// TwinCAT 3 PLC project PLC_Ladder_Hardware_Integration
// ProgramVersion: 3.1.4024.0
// CompilerDefines: VISU_USEWSTRING
// libraries:
//   Tc2_Math, * (Beckhoff Automation GmbH)
//   Tc2_MC2, * (Beckhoff Automation GmbH)
//   Tc2_NC, * (Beckhoff Automation GmbH)
//   Tc2_Standard, * (Beckhoff Automation GmbH)
//   Tc2_System, * (Beckhoff Automation GmbH)
//   Tc2_Utilities, * (Beckhoff Automation GmbH)
//   Tc3_Module, * (Beckhoff Automation GmbH)
// project tree:
//   / GlobalTextList.TcGTLO (not stored), PlcTask.TcTTO, Visualization Manager.TcVMO (not stored)
//   GVLs/ GVL.TcGVL (not stored), GVLLD.TcGVL
//   POUs/ MAIN.TcPOU (not stored), ladder_logic_diagram.TcPOU, Meters_Travelled.TcPOU (not stored), SYSTEM.TcPOU (not stored), Safety_Zones.TcDUT (not stored)
//   VISUs/ Charge_Velocity_Distance.TcVIS (not stored), Header.TcVIS (not stored), ImagePool.TcIPO (not stored), log_file.TcVIS, MainScreen.TcVIS (not stored), Nav.TcVIS, Nav_1.TcVIS, Safty_Zones_and_Modes.TcVIS (not stored)
// real-time tasks:
//   TASK PlcTask: cycle T#10ms, priority 20, ADS port 350
//   TASK VISU_TASK: cycle T#200000us, priority 30, ADS port 351
// motion (NC):
//   TASK NC-Task 1 SAF: cycle T#2ms, priority 4, ADS port 501
//   TASK NC-Task 1 SVB: cycle T#10ms, priority 8, ADS port 511
//   AXIS Axis 1 (id 1)
//     Dynamic: Acceleration=5067.48, Deceleration=5067.48, Jerk=23830.8
//     Velo: RefSearch=14.56175, RefSync=14.56175, SlowManual=72.80875, FastManual=436.8525, Fast=1456.175, Maximum=1456.17
//     TargetPosControl: Range=20
//     OtherSettings: AllowMotionCmdToSlave=true, PulseDistancePos=20, PulseDistanceNeg=20
//     encoder EncType=19
//       EncPara: ScaleFactorNumerator=15.7, ScaleFactorDenominator=1048576, Inverse=true, MaxCount=#xffffffff
//     drive DrvType=16
//       DrvPara: Inverse=true, MaxCount=#xffffffff
//         Analog: VeloReferenz=1601.7925, VeloScale=32, TorqueSetpointScale=10, ScaleFactorActTorque=0.1
//         TimeComp: TaskDelayCycles=1
//     controller CtrType=1
//       CtrPara: PriorControlFactor=1
//         PosDiffControl: Range=40000
//         Observer: BandWidth=20
//   AXIS Axis 2 (id 2)
//     Dynamic: Acceleration=5067.48, Deceleration=5067.48, Jerk=23830.8
//     Velo: RefSearch=14.56175, RefSync=14.56175, SlowManual=72.80875, FastManual=436.8525, Fast=1456.175, Maximum=1456.17
//     TargetPosControl: Range=20
//     OtherSettings: AllowMotionCmdToSlave=true, PulseDistancePos=20, PulseDistanceNeg=20
//     encoder EncType=19
//       EncPara: ScaleFactorNumerator=15.7, ScaleFactorDenominator=1048576, MaxCount=#xffffffff
//     drive DrvType=16
//       DrvPara: MaxCount=#xffffffff
//         Analog: VeloReferenz=1601.7925, VeloScale=32, TorqueSetpointScale=10, ScaleFactorActTorque=0.1
//         TimeComp: TaskDelayCycles=1
//     controller CtrType=1
//       CtrPara: PriorControlFactor=1
//         PosDiffControl: Range=40000
//         Observer: BandWidth=20
//   AXIS Axis 3 (id 3)
//     Dynamic: Acceleration=14588.3136, Deceleration=14588.3136, Jerk=43764.9408
//     Velo: RefSearch=97.255424, RefSync=97.255424, SlowManual=486.27712, FastManual=2917.66272, Fast=9725.5424, Maximum=9725.5424
//     OtherSettings: AllowMotionCmdToSlave=true
//     encoder EncType=19
//       EncPara: ScaleFactorNumerator=104.8576, ScaleFactorDenominator=1048576, MaxCount=#xffffffff
//     drive DrvType=16
//       DrvPara: MaxCount=#xffffffff
//         Analog: VeloReferenz=10698.09664, VeloScale=32, TorqueSetpointScale=10, ScaleFactorActTorque=0.1
//         TimeComp: TaskDelayCycles=1
//     controller CtrType=1
//       CtrPara: PriorControlFactor=1
//         PosDiffControl: Range=10
//         Observer: BandWidth=20
// variable links:
//   PLC_Ladder_Hardware_Integration/PLC_Ladder_Hardware_Integration Instance <-> NC-Task 1 SAF/Axes/Axis 1
//     PlcTask Inputs/MAIN.AxisB.NcToPlc <-> Outputs/ToPlc
//     PlcTask Outputs/MAIN.AxisB.PlcToNc <-> Inputs/FromPlc
//   PLC_Ladder_Hardware_Integration/PLC_Ladder_Hardware_Integration Instance <-> NC-Task 1 SAF/Axes/Axis 2
//     PlcTask Inputs/MAIN.AxisA.NcToPlc <-> Outputs/ToPlc
//     PlcTask Outputs/MAIN.AxisA.PlcToNc <-> Inputs/FromPlc

CONFIGURATION PLC_Ladder_Hardware_Integration
    RESOURCE PLC ON TwinCAT3
        TASK PlcTask(INTERVAL := T#10ms, PRIORITY := 20);
        PROGRAM ladder_logic_diagram WITH PlcTask : ladder_logic_diagram;
        PROGRAM MAIN WITH PlcTask : MAIN;
    END_RESOURCE
END_CONFIGURATION

// ---- GVLs/GVLLD.TcGVL
{attribute 'qualified_only'}
VAR_GLOBAL
	
//Input Variables 
ONOFF_Buton               AT %I* : BOOL;
Manual_Stop_Buton         AT %I* : BOOL;
Manual_Mode_Buton         AT %I* : BOOL;
Autonomous_Mode_Buton     AT %I* : BOOL;
Lock_Mode_Buton           AT %I* : BOOL;
Clear_Reset_Buton         AT %I* : BOOL;
Resume_Buton              AT %I* : BOOL;
view_safety               AT %I* : BOOL;


//Output Variables 
Brake                     AT %Q* : BOOL;  
Kontak                    AT %Q* : BOOL;
Front_White_Zone          AT %Q* : BOOL;
Front_Red_Zone            AT %Q* : BOOL;
Front_Purple_Zone         AT %Q* : BOOL;
Front_Grey_Pink_Zone      AT %Q* : BOOL;
Robot_Clear_Lidar         AT %Q* : BOOL;
Robot_Manual_Mode         AT %Q* : BOOL;
Robot_Autonomous_Mode     AT %Q* : BOOL;
Robot_Lock_Mode           AT %Q* : BOOL;
Robot_Mode_Run            AT %Q* : BOOL;
lift_up_Q                 AT %Q* : BOOL;
lift_down_Q            	  AT %Q* : BOOL;
zone_1                    AT %Q* : BOOL;
zone_2                    AT %Q* : BOOL;
zone_3                    AT %Q* : BOOL;
zone_4                    AT %Q* : BOOL;
zone_5                    AT %Q* : BOOL;
zone_6                    AT %Q* : BOOL;
auto_charge_signal        AT %Q* : BOOL;

//Memery Variables 

System_Trig               AT %M* : BOOL;
System_Set                AT %M* : BOOL;
Memory_Set		          AT %M* : BOOL;
White                     AT %M* : BOOL;
Red                       AT %M* : BOOL;
Purple                    AT %M* : BOOL;
Grey_Pink                 AT %M* : BOOL;
Lock_Mode_Reset           AT %M* : BOOL;
lift_up           		  AT %M* : BOOL;
lift_down				  AT %M* : BOOL;
lift_stop				  AT %M* : BOOL;
elavator_up				  AT %M* : BOOL;
elavator_down			  AT %M* : BOOL;
auto_charge_on            AT %M* : BOOL;
auto_charge_off           AT %M* : BOOL;
view_safety_state         AT %M* : BOOL;

first_time_read           AT %M* : BOOL;
second_time_read          AT %M* : BOOL;
END_VAR

// ---- POUs/ladder_logic_diagram.TcPOU
PROGRAM ladder_logic_diagram 
VAR
	t2s: TIME := TIME#3S;
	t0s: TIME := TIME#0S;
	Timer: TON;
	input : BOOL;
	output : BOOL; 
	TON_Reset: TON;
	TON_set: TON;
	TON_0: TON;
	TON_Trig: TON;
	TON_Autonomous: TON;
	TON_Manual: TON;
	TON_Lock: TON;
	Robot_Mode_Timer: TON;
	liftUP: TON;
	liftDOWN: TON;
	load_button  AT %I* : BOOL ;
	load_active AT %Q*: BOOL;
	trigger AT %M* : BOOL ;
	T: TIME;
	TON_1: TON;
	TON2: TON;
	TON_3: TON;
	activate_time_read: BOOL;
	TON_4: TON;
	second_read_triggered: BOOL;
	first_read_triggered: BOOL;
	TON_5: TON;
	TON_6: TON;
	TON_7: TON;
END_VAR
VAR // added by the converter: edge detectors and wires of the graphical bodies
    _rt1 : R_TRIG;
    _w1 : BOOL;
END_VAR

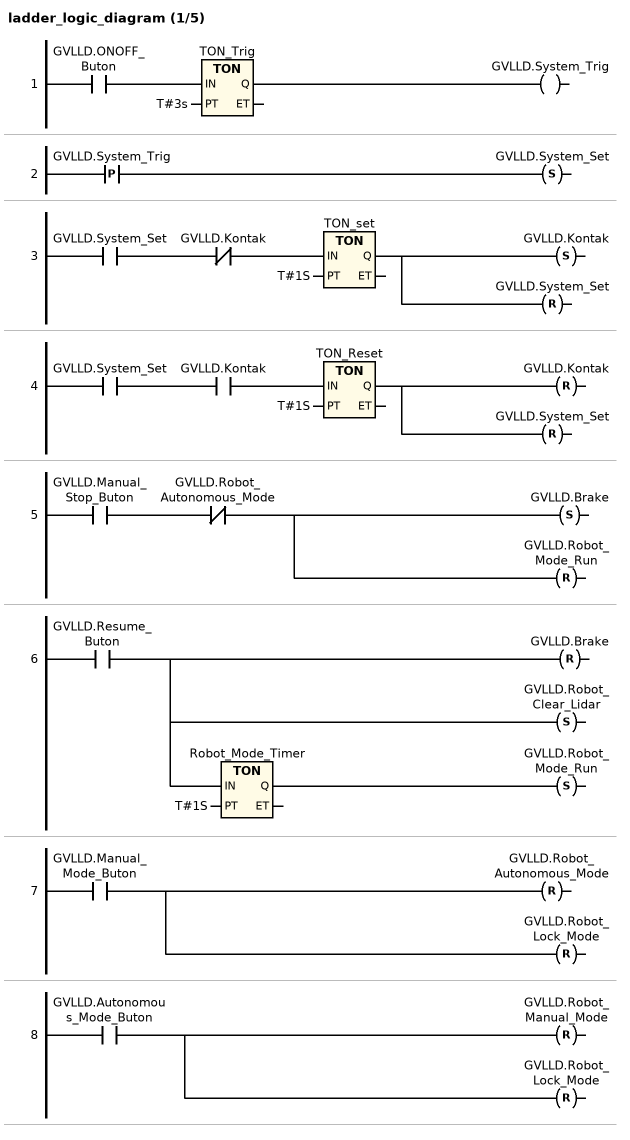
// NETWORK 1
TON_Trig(IN := GVLLD.ONOFF_Buton, PT := T#3s); // TON
GVLLD.System_Trig := TON_Trig.Q;

// NETWORK 2
_rt1(CLK := GVLLD.System_Trig);
GVLLD.System_Set S= _rt1.Q;

// NETWORK 3
TON_set(IN := GVLLD.System_Set AND NOT GVLLD.Kontak, PT := T#1S); // TON
GVLLD.Kontak S= TON_set.Q;
GVLLD.System_Set R= TON_set.Q;

// NETWORK 4
TON_Reset(IN := GVLLD.System_Set AND GVLLD.Kontak, PT := T#1S); // TON
GVLLD.Kontak R= TON_Reset.Q;
GVLLD.System_Set R= TON_Reset.Q;

// NETWORK 5
_w1 := GVLLD.Manual_Stop_Buton AND NOT GVLLD.Robot_Autonomous_Mode;
GVLLD.Brake S= _w1;
GVLLD.Robot_Mode_Run R= _w1;

// NETWORK 6
GVLLD.Brake R= GVLLD.Resume_Buton;
GVLLD.Robot_Clear_Lidar S= GVLLD.Resume_Buton;
Robot_Mode_Timer(IN := GVLLD.Resume_Buton, PT := T#1S); // TON
GVLLD.Robot_Mode_Run S= Robot_Mode_Timer.Q;

// NETWORK 7
GVLLD.Robot_Autonomous_Mode R= GVLLD.Manual_Mode_Buton;
GVLLD.Robot_Lock_Mode R= GVLLD.Manual_Mode_Buton;

// NETWORK 8
GVLLD.Robot_Manual_Mode R= GVLLD.Autonomous_Mode_Buton;
GVLLD.Robot_Lock_Mode R= GVLLD.Autonomous_Mode_Buton;

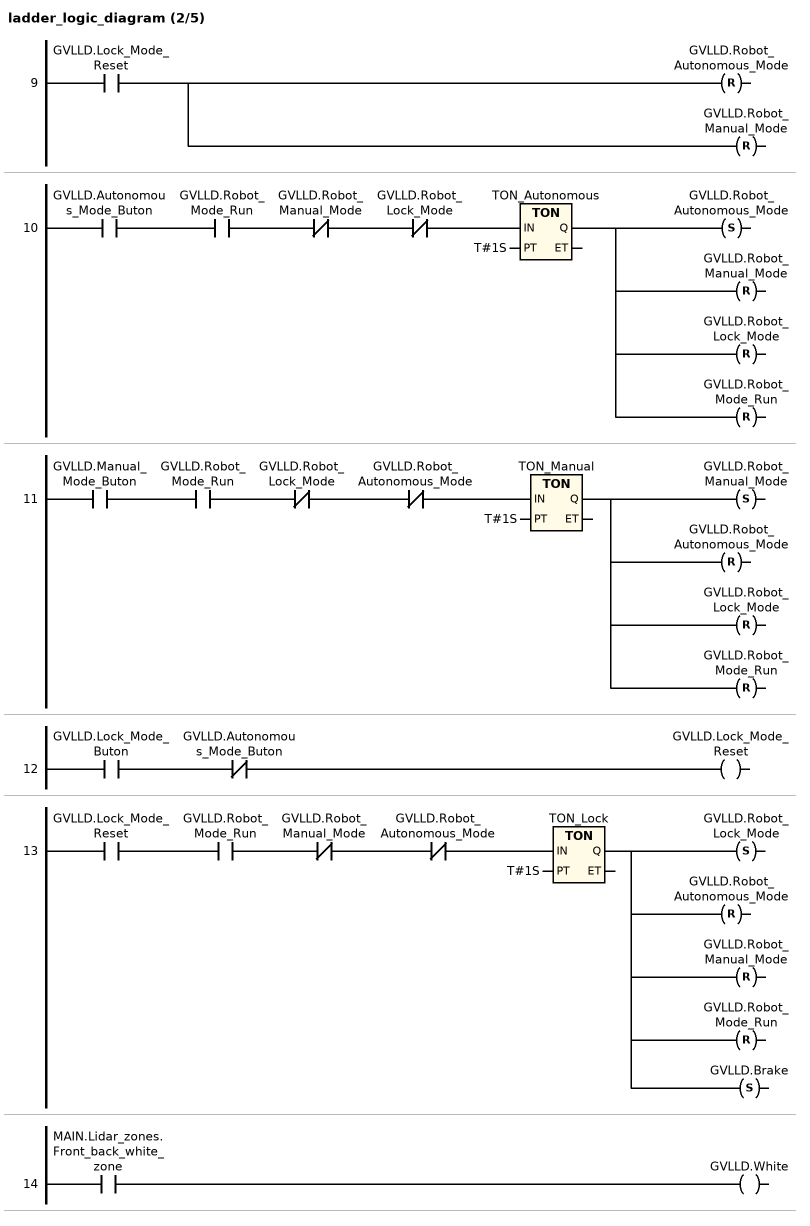
// NETWORK 9
GVLLD.Robot_Autonomous_Mode R= GVLLD.Lock_Mode_Reset;
GVLLD.Robot_Manual_Mode R= GVLLD.Lock_Mode_Reset;

// NETWORK 10
TON_Autonomous(IN := GVLLD.Autonomous_Mode_Buton AND GVLLD.Robot_Mode_Run AND NOT GVLLD.Robot_Manual_Mode AND NOT GVLLD.Robot_Lock_Mode, PT := T#1S); // TON
GVLLD.Robot_Autonomous_Mode S= TON_Autonomous.Q;
GVLLD.Robot_Manual_Mode R= TON_Autonomous.Q;
GVLLD.Robot_Lock_Mode R= TON_Autonomous.Q;
GVLLD.Robot_Mode_Run R= TON_Autonomous.Q;

// NETWORK 11
TON_Manual(IN := GVLLD.Manual_Mode_Buton AND GVLLD.Robot_Mode_Run AND NOT GVLLD.Robot_Lock_Mode AND NOT GVLLD.Robot_Autonomous_Mode, PT := T#1S); // TON
GVLLD.Robot_Manual_Mode S= TON_Manual.Q;
GVLLD.Robot_Autonomous_Mode R= TON_Manual.Q;
GVLLD.Robot_Lock_Mode R= TON_Manual.Q;
GVLLD.Robot_Mode_Run R= TON_Manual.Q;

// NETWORK 12
GVLLD.Lock_Mode_Reset := GVLLD.Lock_Mode_Buton AND NOT GVLLD.Autonomous_Mode_Buton;

// NETWORK 13
TON_Lock(IN := GVLLD.Lock_Mode_Reset AND GVLLD.Robot_Mode_Run AND NOT GVLLD.Robot_Manual_Mode AND NOT GVLLD.Robot_Autonomous_Mode, PT := T#1S); // TON
GVLLD.Robot_Lock_Mode S= TON_Lock.Q;
GVLLD.Robot_Autonomous_Mode R= TON_Lock.Q;
GVLLD.Robot_Manual_Mode R= TON_Lock.Q;
GVLLD.Robot_Mode_Run R= TON_Lock.Q;
GVLLD.Brake S= TON_Lock.Q;

// NETWORK 14
GVLLD.White := MAIN.Lidar_zones.Front_back_white_zone;

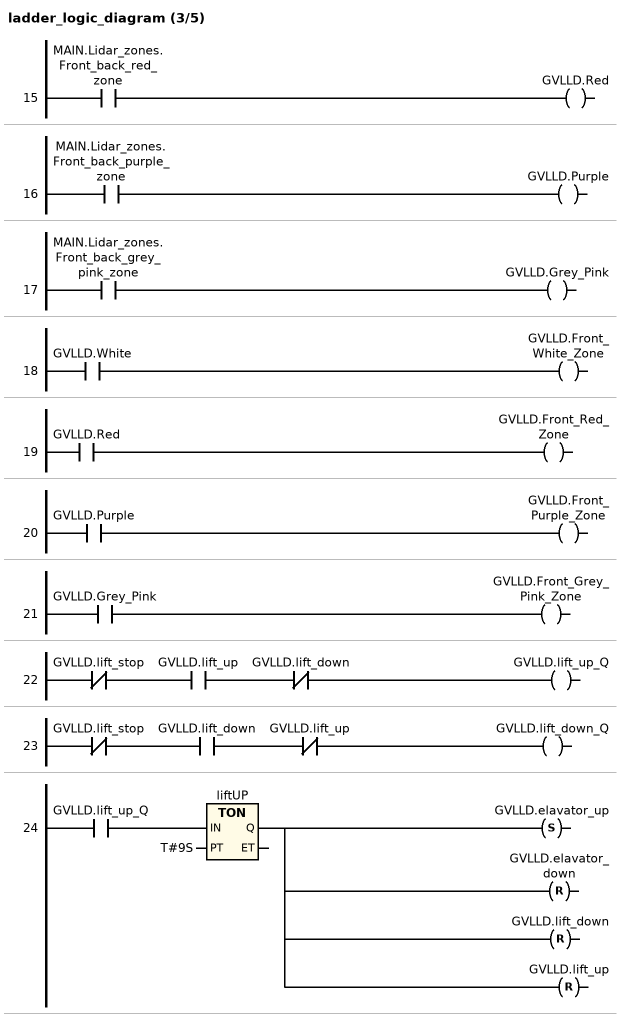
// NETWORK 15
GVLLD.Red := MAIN.Lidar_zones.Front_back_red_zone;

// NETWORK 16
GVLLD.Purple := MAIN.Lidar_zones.Front_back_purple_zone;

// NETWORK 17
GVLLD.Grey_Pink := MAIN.Lidar_zones.Front_back_grey_pink_zone;

// NETWORK 18
GVLLD.Front_White_Zone := GVLLD.White;

// NETWORK 19
GVLLD.Front_Red_Zone := GVLLD.Red;

// NETWORK 20
GVLLD.Front_Purple_Zone := GVLLD.Purple;

// NETWORK 21
GVLLD.Front_Grey_Pink_Zone := GVLLD.Grey_Pink;

// NETWORK 22
GVLLD.lift_up_Q := NOT GVLLD.lift_stop AND GVLLD.lift_up AND NOT GVLLD.lift_down;

// NETWORK 23
GVLLD.lift_down_Q := NOT GVLLD.lift_stop AND GVLLD.lift_down AND NOT GVLLD.lift_up;

// NETWORK 24
liftUP(IN := GVLLD.lift_up_Q, PT := T#9S); // TON
GVLLD.elavator_up S= liftUP.Q;
GVLLD.elavator_down R= liftUP.Q;
GVLLD.lift_down R= liftUP.Q;
GVLLD.lift_up R= liftUP.Q;

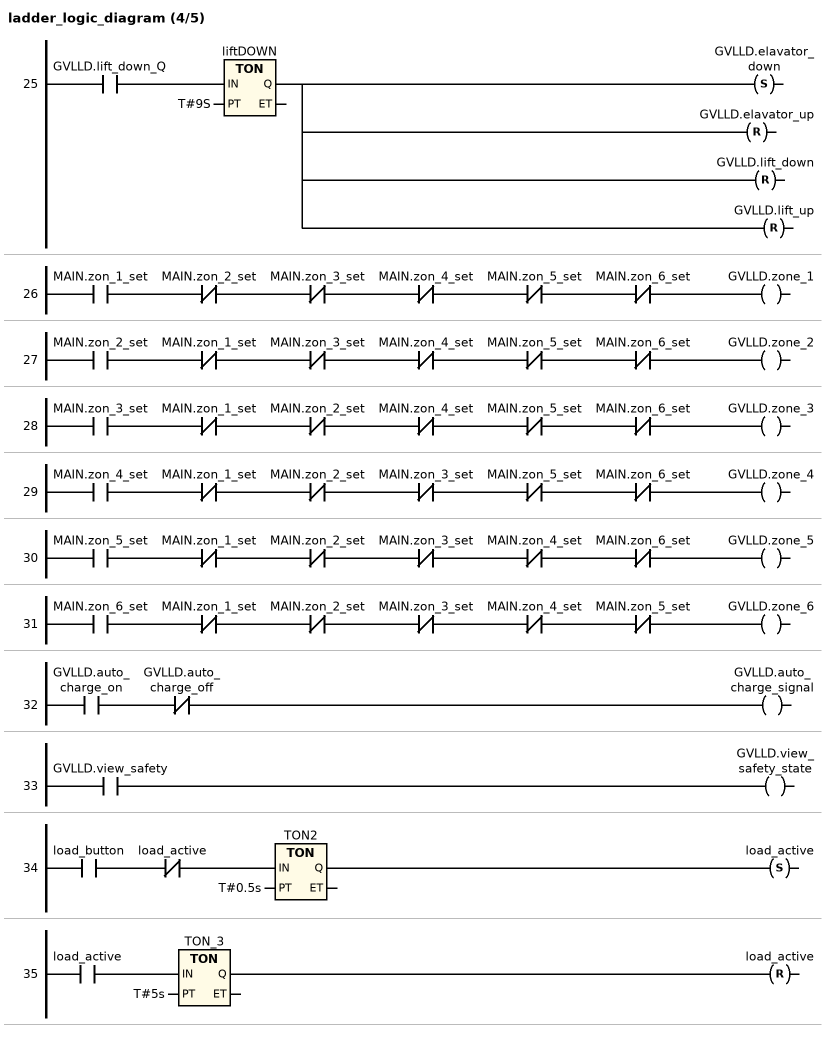
// NETWORK 25
liftDOWN(IN := GVLLD.lift_down_Q, PT := T#9S); // TON
GVLLD.elavator_down S= liftDOWN.Q;
GVLLD.elavator_up R= liftDOWN.Q;
GVLLD.lift_down R= liftDOWN.Q;
GVLLD.lift_up R= liftDOWN.Q;

// NETWORK 26
GVLLD.zone_1 := MAIN.zon_1_set AND NOT MAIN.zon_2_set AND NOT MAIN.zon_3_set AND NOT MAIN.zon_4_set AND NOT MAIN.zon_5_set AND NOT MAIN.zon_6_set;

// NETWORK 27
GVLLD.zone_2 := MAIN.zon_2_set AND NOT MAIN.zon_1_set AND NOT MAIN.zon_3_set AND NOT MAIN.zon_4_set AND NOT MAIN.zon_5_set AND NOT MAIN.zon_6_set;

// NETWORK 28
GVLLD.zone_3 := MAIN.zon_3_set AND NOT MAIN.zon_1_set AND NOT MAIN.zon_2_set AND NOT MAIN.zon_4_set AND NOT MAIN.zon_5_set AND NOT MAIN.zon_6_set;

// NETWORK 29
GVLLD.zone_4 := MAIN.zon_4_set AND NOT MAIN.zon_1_set AND NOT MAIN.zon_2_set AND NOT MAIN.zon_3_set AND NOT MAIN.zon_5_set AND NOT MAIN.zon_6_set;

// NETWORK 30
GVLLD.zone_5 := MAIN.zon_5_set AND NOT MAIN.zon_1_set AND NOT MAIN.zon_2_set AND NOT MAIN.zon_3_set AND NOT MAIN.zon_4_set AND NOT MAIN.zon_6_set;

// NETWORK 31
GVLLD.zone_6 := MAIN.zon_6_set AND NOT MAIN.zon_1_set AND NOT MAIN.zon_2_set AND NOT MAIN.zon_3_set AND NOT MAIN.zon_4_set AND NOT MAIN.zon_5_set;

// NETWORK 32
GVLLD.auto_charge_signal := GVLLD.auto_charge_on AND NOT GVLLD.auto_charge_off;

// NETWORK 33
GVLLD.view_safety_state := GVLLD.view_safety;

// NETWORK 34
TON2(IN := load_button AND NOT load_active, PT := T#0.5s); // TON
load_active S= TON2.Q;

// NETWORK 35
TON_3(IN := load_active, PT := T#5s); // TON
load_active R= TON_3.Q;

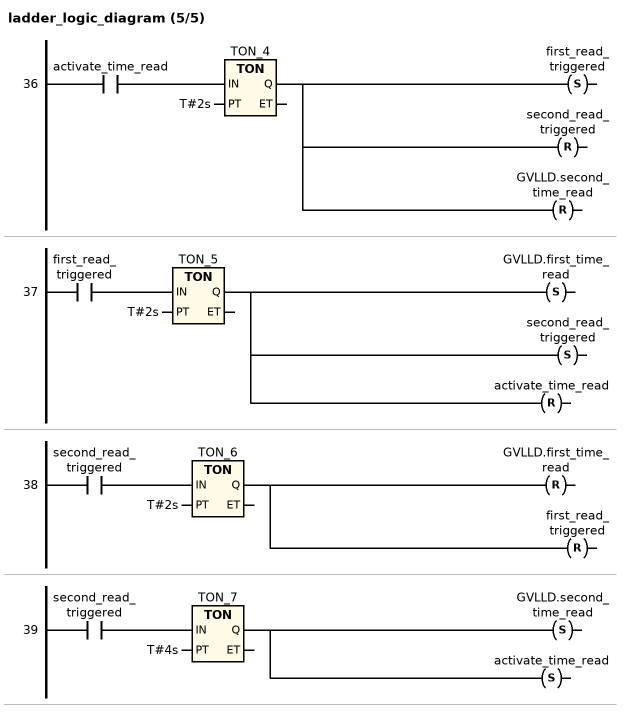
// NETWORK 36
TON_4(IN := activate_time_read, PT := T#2s); // TON
first_read_triggered S= TON_4.Q;
second_read_triggered R= TON_4.Q;
GVLLD.second_time_read R= TON_4.Q;

// NETWORK 37
TON_5(IN := first_read_triggered, PT := T#2s); // TON
GVLLD.first_time_read S= TON_5.Q;
second_read_triggered S= TON_5.Q;
activate_time_read R= TON_5.Q;

// NETWORK 38
TON_6(IN := second_read_triggered, PT := T#2s); // TON
GVLLD.first_time_read R= TON_6.Q;
first_read_triggered R= TON_6.Q;

// NETWORK 39
TON_7(IN := second_read_triggered, PT := T#4s); // TON
GVLLD.second_time_read S= TON_7.Q;
activate_time_read S= TON_7.Q;

END_PROGRAM

// ---- VISUs/log_file.TcVIS
VISUALIZATION log_file  // 2x2
END_VISUALIZATION

// ---- VISUs/Nav.TcVIS
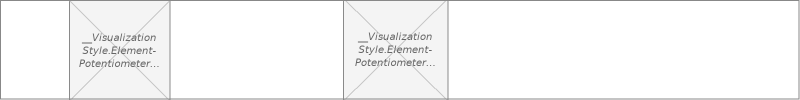
VISUALIZATION Nav  // 800x100
    Image (343,-2 105x103)
    Image (69,0 101x101)
        OnMouseDown: change screen: Safty_Zones_and_Modes
END_VISUALIZATION

// ---- VISUs/Nav_1.TcVIS
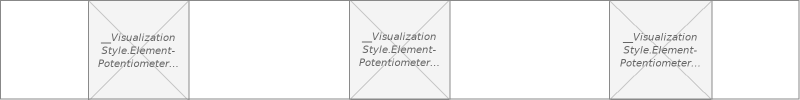
VISUALIZATION Nav_1  // 800x100
    Image (609,0 103x100)
        OnMouseDown: change screen: Charge_Velocity_Distance
    Image (88,0 101x101)
        OnMouseDown: change screen: Safty_Zones_and_Modes
    Image (349,-1 101x101)
        OnMouseDown: change screen: MainScreen
END_VISUALIZATION
